# EPICS autosave request: ADEuresys/EuresysApp/Db/Euresys_settings.req
file "ADGenICam_settings.req", P=$(P), R=$(R)
$(P)$(R)TimeStampMode
$(P)$(R)UniqueIdMode
$(P)$(R)ConvertPixelFormat
$(P)$(R)UnpackingMode
